FUNCTION_BLOCK fbTaskPiotrUN EXTENDS fbUN
VAR
	// Arrays with 'em' universal structure and 'fbEM' containing ST_MACHINE structure which contains of references to fbEM function block
	em : ARRAY[1..Counters.packmlEmLast] OF ST_EM;
	fbEM : ARRAY[1..Counters.packmlEmLast] OF ST_MACHINE;
	
	// Array containing all instances fo fbSliderEM with its own iterator
	SliderEM : ARRAY[1..Counters.SliderEMNo] OF fbSliderEM;
	iSliderEM : DINT := 1;
	
	// Array containing all instances fo fbSliderWithGripperEM with its own iterator
	SliderWithGripperEM : ARRAY[1..Counters.SliderWithGripperEMNo] OF fbSliderWithGripperEM;
	iSliderWithGripperEM : DINT := 1;
	
	// Array containing all instances fo fbXYMoverEM with its own iterator
	XYMoverEM : ARRAY[1..Counters.XYMoverEMNo] OF fbXYMoverEM;
	iXYMoverEM : DINT := 1;
	
	i : DINT;
	State : INT := 0;
	declareIterator : DINT;
	moduleWorkIterator : DINT;
	initialConfig: BOOL := TRUE;
END_VAR

// fbEM and em array number:
// 1 <- XYMovers
// 2 <- SliderWithGripper
// 3 <- XYMover
// 4 <- Slider
// 5 <- Slider

////////////////////////////////////////////////////////////////////////////////////////////////////////////////////////////
// All init configuration done here
IF initialConfig THEN
	initialConfig := FALSE;
	// Specifing module type of each module in array
	em[1].Config.Functionality := E_Function.eXYMover;
	em[2].Config.Functionality := E_Function.eSliderWithGripper;
	em[3].Config.Functionality := E_Function.eXYMover;
	em[4].Config.Functionality := E_Function.eSlider;
	em[5].Config.Functionality := E_Function.eSlider;

	// FOR loop to specify config for each module
	FOR declareIterator := 1 TO Counters.packmlEmLast DO
		em[declareIterator].Config.Data.I REF= GVL.aInput[declareIterator];
		em[declareIterator].Config.Data.Q REF= GVL.aOutput[declareIterator];

		CASE em[declareIterator].Config.Functionality OF
			E_Function.eSlider:
				fbEM[declareIterator].fbEM REF= SliderEM[iSliderEM];
				iSliderEM := iSliderEM + 1;
			E_Function.eSliderWithGripper:
				fbEM[declareIterator].fbEM REF= SliderWithGripperEM[iSliderWithGripperEM];
				iSliderWithGripperEM := iSliderWithGripperEM + 1;
			E_Function.eXYMover:
				fbEM[declareIterator].fbEM REF= XYMoverEM[iXYMoverEM];
				iXYMoverEM := iXYMoverEM + 1;
		END_CASE
	END_FOR
END_IF

////////////////////////////////////////////////////////////////////////////////////////////////////////////////////////////
// Modules work loop (idk yet if is better to have it at the beggining or bottom of UN)
FOR moduleWorkIterator := 1 TO Counters.packmlEmLast DO
	fbEM[moduleWorkIterator].fbEM(em := em[moduleWorkIterator], un := un, EnableSim := EnableSim, CmdSim := FALSE);
END_FOR

////////////////////////////////////////////////////////////////////////////////////////////////////////////////////////////


IF cell.Cmd = E_CMD_CELL.STOP AND NOT (State = 100 OR State = 110) THEN
	State := 1000;
END_IF

IF cell.Cmd = E_CMD_CELL.ABORT AND NOT (State = 200 OR State = 210) THEN
	State := 2000;
END_IF

CASE State OF
	0:	un.Status := E_Status.undefined;
		em[2].Config.Data.pick_pos := 3;
		em[2].Config.Data.drop_pos := 2;
		State := 5;
		
	2:	
	
	5:	// Waiting for every EM to become idle state
		FOR i := 1 TO Counters.packmlEmLast DO
			IF NOT (em[i].Status = E_Status.idle) THEN
				un.Cmd := E_CMD.reset;
				RETURN;
			END_IF
		END_FOR
		un.Status := E_Status.idle;
		State := 10;
	
	10:	IF cell.Cmd = E_CMD_CELL.START THEN
			un.Cmd := E_CMD.start;
			un.Status := E_Status.starting;
			State := 20;
		END_IF
	
	20:	// Waiting for every EM to be in execute or starting state
		FOR i := 1 TO Counters.packmlEmLast DO
			IF NOT (em[i].Status = E_Status.execute OR em[i].Status = E_Status.starting) THEN
				RETURN;
			END_IF
		END_FOR
		State := 30;
		
	30:	// Start of my specific task (all modules stays in execute)
		// input -> XY1 -> SWG -> XY2 -> S1 -> SWG -> S2 -> output
		IF em[1].SequenceStep = 20		// XY1
		AND cell.PlaceObject			// Object input signal 
		THEN
			cell.PlaceObject := FALSE;
			em[1].Config.Data.I[5] := TRUE;
			State := 40;
		END_IF
		
	40:	// XY1 -> SWG -> XY2 -> S1 -> SWG -> S2 -> output
		IF em[1].SequenceStep = 60		// XY1
		AND em[2].SequenceStep = 40		// SWG
		THEN
			em[1].Config.Data.I[5] := FALSE;
			em[2].Config.Data.I[3] := TRUE;
			State := 50;
		END_IF
		
	50: // SWG -> XY2 -> S1 -> SWG -> S2 -> output
		IF em[2].SequenceStep = 43		// SWG
		AND em[3].SequenceStep = 20		// XY2
		THEN
			em[2].Config.Data.I[3] := FALSE;
			em[3].Config.Data.I[5] := TRUE;
			State := 60;
		END_IF
		
	60: // XY2 -> S1 -> SWG -> S2 -> output
		em[2].Config.Data.drop_pos := 1;
		em[2].Config.Data.pick_pos := 4;
		IF em[2].SequenceStep = 40		// SWG
		AND em[3].SequenceStep = 60		// XY2
		AND em[4].SequenceStep = 50		// S1
		THEN
			em[3].Config.Data.I[5] := FALSE;
			em[4].Config.Data.I[3] := TRUE;
			State := 70;
		END_IF
		
	70:	// S1 -> SWG -> S2 -> output
		IF em[4].SequenceStep = 70		// S1
		THEN
			em[2].Config.Data.I[3] := TRUE;// SWG
			em[4].Config.Data.I[3] := FALSE;
			State := 80;
		END_IF
		
	80:	// SWG -> S2 -> output
		IF em[2].SequenceStep = 43		// SWG
		AND em[5].SequenceStep = 50		// S2
		THEN
			em[2].Config.Data.I[3] := FALSE;
			em[2].Config.Data.pick_pos := 3;
			em[5].Config.Data.I[3] := TRUE;
			State := 90;
		END_IF
		
	90:	// S2 -> output
		em[2].Config.Data.pick_pos := 3;
		em[2].Config.Data.drop_pos := 2;
		State := 30;

	1000:
		un.Cmd := E_CMD.stop;
		un.Status := E_Status.stopping;
		State := 1010;
	
	1010:
		FOR i := 1 TO Counters.packmlEmLast DO
			IF NOT (em[i].Status = E_Status.stopped) THEN
				un.Status := E_Status.stopped;
				State := 5;
			END_IF
		END_FOR
	
	2000:
		un.Cmd := E_CMD.abort;
		un.Status := E_Status.aborting;
		State := 2010;
	
	2010:
		FOR i := 1 TO Counters.packmlEmLast DO
			IF NOT (em[i].Status = E_Status.aborted) THEN
				;
			ELSE
				State := 2020;
			END_IF
		END_FOR
	
	2020:
		un.Cmd := E_CMD.clear;
		State := 5;
END_CASE

END_FUNCTION_BLOCK

(* stored: Version 1.1.0.1, ProductVersion 3.1.4024.12
   POU fbTaskPiotrUN: Id {e4410345-6b08-4ef7-a94f-07fca8e2946d}, SpecialFunc None *)
